// SIMATIC S7-200 project (STEP 7-Micro/WIN), CPU 224 REL 01.21

SYMBOL_TABLE USR1
手自动              I0.5     // V120.0
主轴启动             I0.7     // V121.4
主轴停              I0.0     // V121.5
复位               I0.2     // V120.1
制动               I0.3     // V120.2
左行               I0.4     // V121.0
右行               I0.6     // V121.1
进刀               I1.0     // V121.2
退刀               I0.1     // V121.3
阶梯锥的长度           VD614    // VD200
记录横向步数           VD570    // VW500
第一段半径            VD252
第二段半径            VD256
第三段半径            VD260
圆弧半径             VD240
进刀量的理论值          VD620
物件半径             VD208
圆台高度             VD232
斜率               VD236
圆台的小半径           VD296
最大进刀量            VD98     // vb101    vd204
圆弧的长度            VD244
实际进刀量            VW520
片选               Q2.2
时钟               Q2.1
数据               Q2.3
最进刀量             VW206
END_SYMBOL_TABLE

ORGANIZATION_BLOCK 主:OB1
TITLE=PLC程序操控一台数控车床，实现圆锥、阶梯锥和圆弧等复杂零件的加工。主程序循环OB1协调各个模块，操作员输入加工参数后，程序通过子程序完成加工路径计算和机床运动控制。设备：主电机、横向电机、纵向电机、传感器、按钮和数显设备 
// 系统通过启动按钮启动加工过程，操作员可通过手动/自动切换开关选择手动或自动模式。在自动模式下，按下启动按钮时，主轴运行输出被激活，主轴电机开始运行，但若按下停止按钮或制动按钮，主轴运行输出会立即关闭，确保加工过程可随时安全中止。
// 加工过程中，横向电机的移动由左行按钮和右行按钮控制。当按下左行按钮时，左行标志置位；当按下右行按钮时，右行标志置位。横向电机左行输出直接由左行标志控制，当左行标志置位时激活；横向电机右行输出直接由右行标志控制，当右行标志置位时激活。横向移动计时器周期性触发，更新横向位置计数器，记录当前的横向位置。
// 纵向电机的进退刀由进刀按钮和退刀按钮控制。按下进刀按钮时，进刀标志置位，驱动纵向电机进刀输出使刀具向前移动；按下退刀按钮时，退刀标志置位，驱动纵向电机退刀输出使刀具后退。纵向移动计时器触发时，更新实际进刀量计数器，记录进刀深度。
// 当需要加工复杂零件时，系统根据加工标志调用相应子程序。例如，加工圆锥时，程序读取圆台高度和物件半径，计算进刀量的理论值，并驱动电机按计算路径移动。进刀量的理论值在加工标志置位时更新，基于圆台高度和物件半径精确计算，确保加工精度。
// 若操作员按下复位按钮，且切换开关处于手动模式，系统会清零横向位置计数器和实际进刀量计数器，恢复到初始状态，为下一次加工做好准备。通过加工计时器和延时启动计时器的协调，程序确保各电机按正确时序启动和停止，实现高效、安全的加工流程。
// 
BEGIN
Network 1 // 网络题目 (单行)
//  
// 网络注释
//  
// 
LD     SM0.1
LPS
MOVB   16#49, SMB30
AENO
ATCH   INT_0:INT0, 8
LRD
MOVD   &VB999, VD10
AENO
MOVD   VD10, VD16
LPP
MOVW   +0, VW14
AENO
ENI
Network 2
LD     SM0.7
=      SM30.0
Network 3
LD     M0.0
TON    T35, +10
Network 4
LD     T35
AW>=   VW14, +7
AW=    VW1000, 16#5657
AW=    VW1005, 16#1003
AB=    VB1004, 1
CALL   通讯一:SBR2
Network 5
LD     T35
AW>=   VW14, +7
AD=    VD1000, 16#52454144
AW=    VW1005, 16#1003
AB=    VB1004, 1
CALL   通讯二:SBR3
Network 6
LD     T35
R      M0.0, 1
MOVW   +0, VW14
MOVD   VD10, VD16
Network 7
LD     SM0.1
MOVB   16#11, VB0
AENO
MOVB   16#11, VB1
Network 8
LD     复位:I0.2
AN     手自动:I0.5
LD     V120.1
AN     V120.0
OLD
O      M4.1
LPS
MOVW   +0, VW500
AENO
MOVW   +0, 实际进刀量:VW520
LRD
MOVW   +20, VW2008
AENO
MOVW   +20, VW2004
LPP
MOVW   +0, VW700
AENO
R      M4.0, 2
Network 9
LD     V120.0
A      手自动:I0.5
EU
LD     主轴启动:I0.7
EU
OLD
LD     V121.4
EU
OLD
O      Q0.4
AN     V121.5
AN     V120.2
AN     制动:I0.3
AN     主轴停:I0.0
=      Q0.4
=      V123.4
Network 10
LDN    退刀:I0.1
AN     进刀:I1.0
AN     右行:I0.6
AN     左行:I0.4
AN     手自动:I0.5
=      M4.2
Network 11
LDN    V121.2
AN     V120.0
AN     V121.3
AN     V121.0
AN     V121.1
=      M4.3
Network 12 // 延时启动横纵电机
// 
// 
LD     V120.0
A      手自动:I0.5
A      Q0.4
TON    T39, +30
Network 13 // 横向时钟
// 
// 
LD     SM0.0
LPS
AN     M0.4
TON    T32, VW632
LPP
A      T32
=      M0.4
Network 14 // 左行
// 
// 
LD     左行:I0.4
O      V121.0
AN     V120.0
AN     手自动:I0.5
LD     T39
A      M3.0
OLD
AN     V120.2
AN     制动:I0.3
=      V123.0
Network 15
LD     T32
A      V123.0
RRB    VB0, 1
AENO
INCW   VW500
Network 16 // 右行
// 
// 
LD     右行:I0.6
O      V121.1
AN     V120.0
AN     手自动:I0.5
LD     T39
A      M3.1
OLD
AN     V120.2
AN     制动:I0.3
=      V123.1
Network 17
LD     T32
A      V123.1
RLB    VB0, 1
AENO
DECW   VW500
Network 18
LDN    M4.2
ON     M4.3
LPS
A      V0.0
=      Q0.0
LRD
A      V0.1
=      Q0.1
LRD
A      V0.2
=      Q0.2
LPP
A      V0.3
=      Q0.3
Network 19
LD     SM0.0
LPS
ITD    VW500, VD502
AENO
DTR    VD502, VD550
LPP
MOVR   VD550, 记录横向步数:VD570
*R     0.0029166, 记录横向步数:VD570
Network 20 // 进退刀时钟
// 
// 
LD     SM0.0
LPS
AN     M0.2
TON    T96, VW632
LPP
A      T96
=      M0.2
Network 21 // 退刀
// 
// 
LD     退刀:I0.1
O      V121.2
AN     V120.0
AN     手自动:I0.5
LD     T39
A      M3.3
OLD
AN     V120.2
AN     制动:I0.3
=      V123.2
Network 22
LD     T96
A      V123.2
RLB    VB1, 1
AENO
DECW   实际进刀量:VW520
Network 23 // 进刀
// 
// 
LD     进刀:I1.0
O      V121.3
AN     V120.0
AN     手自动:I0.5
LD     T39
A      M3.2
OLD
AN     V120.2
AN     制动:I0.3
=      V123.3
Network 24
LD     T96
A      V123.3
RRB    VB1, 1
AENO
INCW   实际进刀量:VW520
Network 25
LDN    M4.2
ON     M4.3
LPS
A      V1.0
=      Q0.5
LRD
A      V1.1
=      Q0.6
LRD
A      V1.2
=      Q0.7
LPP
A      V1.3
=      Q1.0
Network 26
LDN    M4.0
AN     M3.1
AW<    VW500, VW202
O      V123.7
LPS
AN     V123.7
AN     M3.2
AN     M3.3
=      M3.0
S      M3.6, 1
LRD
LD     V123.6
AW<    实际进刀量:VW520, VW622
LDW<   实际进刀量:VW520, VW2008
AN     V123.6
AW>=   VW622, VW2008
OLD
ALD
=      M3.2
LPP
AW<=   实际进刀量:VW520, VW2008
A      M3.2
A      M3.7
MOVW   VW500, VW600
AENO
R      M3.7, 1
Network 27
LDW>=  VW500, VW202
OW>    实际进刀量:VW520, VW622
LDN    V123.6
A      M3.3
OLD
AW>=   VW500, +1
AW>    实际进刀量:VW520, -4
=      M3.3
R      M3.6, 1
S      M3.4, 1
AW>    VW500, VW700
MOVW   VW500, VW700
Network 28
LDW>=  VW500, VW202
LD     M3.4
AN     V120.5
OLD
AN     V123.6
AN     M3.2
AN     M3.3
LPS
S      M3.1, 1
S      M3.7, 1
A      M3.6
EU
LPS
MOVW   +0, VW600
AENO
S      M4.0, 1
LPP
MOVW   +0, VW2008
AENO
S      V123.6, 1
LPP
EU
MOVW   VW2008, VW2012
+I     最进刀量:VW206, VW2008
AENO
R      M3.4, 1
Network 29
LDW<=  VW500, VW600
R      M3.1, 1
Network 30 // 纵向速度
// 
// 
LD     手自动:I0.5
O      V120.0
AW<    实际进刀量:VW520, VW2012
LD     V123.5
AN     V120.0
OLD
BTI    VB106, VW634
NOT
BTI    VB107, VW634
Network 31 // 横向速度
// 
// 
LD     手自动:I0.5
O      V120.0
AW<=   实际进刀量:VW520, +0
LDN    手自动:I0.5
O      V123.5
AN     V120.0
OLD
BTI    VB104, VW632
NOT
BTI    VB105, VW632
Network 32
LD     V120.4
CALL   圆锥:SBR0
Network 33
LD     V120.5
CALL   园弧:SBR6
Network 34
LD     V120.3
CALL   转换:SBR1
Network 35
LD     V120.6
CALL   阶梯锥:SBR5
Network 36
LD     V123.7
CALL   SBR_7:SBR7
Network 37
LD     SM0.0
CALL   数显:SBR4
END_ORGANIZATION_BLOCK

SUBROUTINE_BLOCK 圆锥:SBR0
TITLE= 
// 子程序注释
// 按 F1 获得帮助及举例程序
//  
BEGIN
Network 1
LD     V120.4
MOVR   圆台高度:VD232, LD0
AENO
/R     0.002916666, LD0
AENO
ROUND  LD0, VD200
Network 2
//  
// 
//  
// 
LD     SM0.0
LPS
MOVR   记录横向步数:VD570, VD558
AENO
*R     斜率:VD236, VD558
AENO
MOVR   圆台的小半径:VD296, VD554
+R     VD558, VD554
LPP
MOVR   物件半径:VD208, VD562
-R     VD554, VD562
Network 3
LD     SM0.0
MOVR   VD562, VD564
AENO
/R     0.00375, VD564
AENO
TRUNC  VD564, 进刀量的理论值:VD620
END_SUBROUTINE_BLOCK

SUBROUTINE_BLOCK 转换:SBR1
TITLE=
BEGIN
Network 1 // 总长度
// 
// 
LD     SM0.0
LPS
MOVD   VD97, LD2
AENO
ANDD   16#FF, LD2
AENO
DTR    LD2, LD6
LPP
MOVR   LD6, LD10
AENO
/R     0.002916666, LD10
AENO
ROUND  LD10, VD200
Network 2 // 最大进到量
// 
// 
LD     SM0.0
LPS
MOVD   最大进刀量:VD98, LD2
AENO
ANDD   16#FF, LD2
AENO
DTR    LD2, LD6
LPP
MOVR   LD6, LD10
AENO
/R     0.0375, LD10
AENO
ROUND  LD10, VD204
Network 3 // 圆锥高度
// 
// 
LD     SM0.0
LPS
BTI    VB108, LW0
AENO
ITD    LW0, LD2
LPP
DTR    LD2, 圆台高度:VD232
Network 4 // （圆锥下底面半径-圆锥上底面半径）/圆台高度
// 
// 
LD     SM0.0
LPS
BTI    VB109, VW710
AENO
BTI    VB124, VW712
LRD
MOVW   VW710, VW714
AENO
-I     VW712, VW714
AENO
ITD    VW714, VD716
LPP
DTR    VD716, VD720
AENO
MOVR   VD720, 斜率:VD236
/R     圆台高度:VD232, 斜率:VD236
Network 5
LD     SM0.0
MOVB   VB109, VB592
AB>    VB109, VB124
MOVB   VB124, VB592
Network 6
LD     SM0.0
LPS
BTI    VB592, LW0
AENO
ITD    LW0, LD2
LPP
DTR    LD2, 圆台的小半径:VD296
Network 7 // 物件半径
// 
// 
LD     SM0.0
LPS
ITD    VW102, LD2
AENO
DTR    LD2, LD6
LPP
MOVR   LD6, 物件半径:VD208
/R     100.0, 物件半径:VD208
Network 8 // 圆弧半径
// 
// 
LD     SM0.0
MOVD   VD107, LD2
AENO
ANDD   16#FF, LD2
AENO
DTR    LD2, VD602
DTR    LD2, 圆弧半径:VD240
Network 9 // 圆弧长度
// 
// 
LD     SM0.0
LPS
MOVD   VD108, LD2
AENO
ANDD   16#7F, LD2
AENO
DTR    LD2, VD606
AENO
SRD    LD2, 1
LRD
DTR    LD2, 圆弧的长度:VD244
LPP
A      V111.7
*R     -1.0, 圆弧的长度:VD244
+R     0.0, 圆弧的长度:VD244
Network 10 // 圆弧起始半径
// 
// 
LD     SM0.0
MOVD   VD109, LD2
AENO
ANDD   16#FF, LD2
AENO
DTR    LD2, VD248
Network 11 // 第一段长度
// 
// 
LD     SM0.0
LPS
MOVR   圆弧半径:VD240, LD6
AENO
-R     圆弧的长度:VD244, LD6
AENO
MOVR   圆弧半径:VD240, LD10
+R     圆弧的长度:VD244, LD10
LRD
MOVR   LD6, LD14
AENO
*R     LD10, LD14
AENO
SQRT   LD14, VD672
LPP
MOVR   VD248, VD676
-R     VD672, VD676
Network 12 // 第一段半径
// 
// 
LD     SM0.0
MOVD   VD110, LD2
AENO
ANDD   16#FF, LD2
AENO
DTR    LD2, 第一段半径:VD252
Network 13 // 第二段半径
// 
// 
LD     SM0.0
MOVD   VD111, LD2
AENO
ANDD   16#FF, LD2
AENO
DTR    LD2, 第二段半径:VD256
Network 14 // 第三段半径
// 
// 
LD     SM0.0
MOVD   VD112, LD2
AENO
ANDD   16#FF, LD2
AENO
DTR    LD2, 第三段半径:VD260
Network 15 // 阶梯锥第一段长
// 
// 
LD     SM0.0
MOVD   VD122, LD2
AENO
ANDD   16#FF, LD2
AENO
DTR    LD2, VD300
Network 16 // 阶梯锥第二段长
// 
// 
LD     SM0.0
MOVD   VD123, LD2
AENO
ANDD   16#FF, LD2
AENO
DTR    LD2, VD304
Network 17 // 阶梯锥第三段长
// 
// 
LD     SM0.0
MOVD   VD124, LD2
AENO
ANDD   16#FF, LD2
AENO
DTR    LD2, VD308
Network 18
LD     SM0.0
MOVR   VD304, VD610
AENO
+R     VD300, VD610
AENO
MOVR   VD610, 阶梯锥的长度:VD614
+R     VD308, 阶梯锥的长度:VD614
Network 19
LD     V120.3
R      V120.3, 1
END_SUBROUTINE_BLOCK

SUBROUTINE_BLOCK 通讯一:SBR2
TITLE=
BEGIN
Network 1
LD     SM0.0
MOVD   &VB100, VD20
ANDD   16#FF, VD999
+D     VD999, VD20
MOVB   VB1003, *VD20
END_SUBROUTINE_BLOCK

SUBROUTINE_BLOCK 通讯二:SBR3
TITLE=
BEGIN
Network 1
LD     SM0.0
MOVD   16#52454144, VD96
MOVW   16#1003, VW150
MOVB   56, VB95
XMT    VB95, 0
END_SUBROUTINE_BLOCK

SUBROUTINE_BLOCK 数显:SBR4
TITLE=
BEGIN
Network 1
LD     SM0.1
LPS
MOVW   16#F9FF, VW3626
AENO
MOVW   16#FAF8, VW3628
AENO
MOVW   16#FBFF, VW3630
AENO
MOVW   16#FCFF, VW3632
LRD
MOVD   &VB3626, AC2
LRD
S      M20.0, 1
LPP
MOVW   VW3626, VW3600
Network 2
LD     SM0.0
MOVD   &VB3632, AC3
Network 3 // 发送程序
//  
// 网络注释
//  
// 
LD     M20.2
=      M20.1
Network 4
LD     C0
=      M20.2
R      M20.0, 1
Network 5
LD     M20.3
SLW    VW3600, 1
Network 6
LD     M20.0
AN     C0
AN     M20.3
=      M20.3
Network 7
LD     M20.3
LD     C0
CTU    C0, +16
Network 8
LDN    T51
A      M20.1
LPS
S      M20.0, 1
AW<    AC2, AC3
+I     +2, AC2
AENO
MOVW   *AC2, VW3600
AENO
MOVW   *AC2, VW3700
LPP
AW>=   AC2, AC3
MOVD   &VB3624, AC2
Network 9
LD     SM0.0
LPS
AN     M20.2
=      片选:Q2.2
LRD
AN     M20.3
=      时钟:Q2.1
LPP
AN     V3600.7
=      数据:Q2.3
Network 10
LD     SM0.0
MOVR   VD550, VD510
AENO
*R     0.2916666, VD510
AENO
TRUNC  VD510, VD514
Network 11
LD     SM0.0
LPS
ITD    实际进刀量:VW520, VD580
AENO
DTR    VD580, VD584
LRD
MOVR   VD584, VD588
AENO
*R     0.375, VD588
AENO
TRUNC  VD588, VD596
LPP
DTI    VD596, VW594
AENO
AW<    VW594, +0
MOVW   +0, VW594
Network 12
LDN    T51
MOVW   VW594, VW3800
AENO
IBCD   VW3800
AENO
MOVW   VW516, VW3802
AENO
IBCD   VW3802
AENO
MOVW   +0, VW3899
Network 13
LD     T51
A      M20.1
LPS
RLD    VD3800, 4
AENO
MOVD   VD3800, VD3804
ANDD   16#F, VD3804
LRD
AB<    VB3900, 8
INCB   VB3900
LRD
MOVD   VD3804, VD3598
AENO
ORD    VD3898, VD3598
AENO
S      M20.0, 1
LRD
LDB=   VB3900, 7
OB=    VB3900, 2
ALD
ORD    16#F0, VD3598
LPP
AB>=   VB3900, 8
LPS
MOVW   VW594, VW3800
AENO
IBCD   VW3800
AENO
MOVW   VW516, VW3802
IBCD   VW3802
LPP
MOVD   +0, VD3898
Network 14
LDN    SM0.1
TON    T51, +50
Network 15
LD     SM0.0
MOVW   VW594, VW116
AENO
MOVW   VW516, VW118
END_SUBROUTINE_BLOCK

SUBROUTINE_BLOCK 阶梯锥:SBR5
TITLE=
BEGIN
Network 1
LD     V120.6
MOVR   阶梯锥的长度:VD614, LD0
AENO
/R     0.002916666, LD0
AENO
ROUND  LD0, VD200
Network 2
LDR<=  记录横向步数:VD570, VD300
MOVR   物件半径:VD208, VD730
-R     第一段半径:VD252, VD730
Network 3
LDR>   记录横向步数:VD570, VD300
AR<=   记录横向步数:VD570, VD610
MOVR   物件半径:VD208, VD730
-R     第二段半径:VD256, VD730
Network 4
LDR>   记录横向步数:VD570, VD610
AR<=   记录横向步数:VD570, 阶梯锥的长度:VD614
MOVR   物件半径:VD208, VD730
-R     第三段半径:VD260, VD730
Network 5
LD     SM0.0
MOVR   VD730, VD734
AENO
/R     0.00375, VD734
AENO
TRUNC  VD734, 进刀量的理论值:VD620
END_SUBROUTINE_BLOCK

SUBROUTINE_BLOCK 园弧:SBR6
TITLE= 
// 子程序注释
// 按 F1 获得帮助及举例程序
//  
VAR
TEMP1:REAL;	// LD0 
TEMP2:DWORD;	// LD4 
END_VAR
BEGIN
Network 1
LD     V120.5
MOVR   VD606, #TEMP1:LD0
AENO
/R     0.002916666, #TEMP1:LD0
AENO
ROUND  #TEMP1:LD0, VD200
Network 2 // 网络题目 (单行)
//  
// 网络注释
//  
// 
LD     SM0.0
LPS
MOVR   记录横向步数:VD570, VD640
AENO
-R     圆弧的长度:VD244, VD640
AENO
MOVR   圆弧半径:VD240, VD644
-R     VD640, VD644
LRD
MOVR   圆弧半径:VD240, VD648
AENO
+R     VD640, VD648
AENO
MOVR   VD648, VD652
*R     VD644, VD652
LPP
SQRT   VD652, VD656
AENO
MOVR   VD656, VD660
+R     VD676, VD660
Network 3
LD     SM0.0
LPS
MOVR   物件半径:VD208, VD664
AENO
-R     VD660, VD664
AENO
MOVR   VD664, VD668
/R     0.00375, VD668
LPP
TRUNC  VD668, 进刀量的理论值:VD620
END_SUBROUTINE_BLOCK

SUBROUTINE_BLOCK SBR_7:SBR7
TITLE= 
// 子程序注释
// 按 F1 获得帮助及举例程序
//  
BEGIN
Network 1 // 网络题目 (单行)
//  
// 网络注释
//  
// 
LD     V123.7
LPS
BTI    VB100, LW0
AENO
ITD    LW0, LD2
LRD
DTR    LD2, VD200
LRD
MOVR   VD200, VD740
AENO
/R     0.00375, VD740
AENO
TRUNC  VD740, 进刀量的理论值:VD620
LPP
BTI    VB107, VW634
AENO
S      V123.6, 1
Network 2
LDW>=  实际进刀量:VW520, VW622
R      V123.6, 2
MOVD   +0, 进刀量的理论值:VD620
END_SUBROUTINE_BLOCK

INTERRUPT_BLOCK INT_0:INT0
TITLE= 
// 中断程序注释
// 按 F1 获得帮助及举例程序
//  
BEGIN
Network 1 // 网络题目 (单行)
//  
// 网络注释
//  
// 
LD     SM0.0
AW<=   VW14, +20
INCD   VD16
INCW   VW14
MOVB   SMB2, *VD16
=      M0.0
END_INTERRUPT_BLOCK
